Universal Robots PolyScope program: ur_comm_test.urp

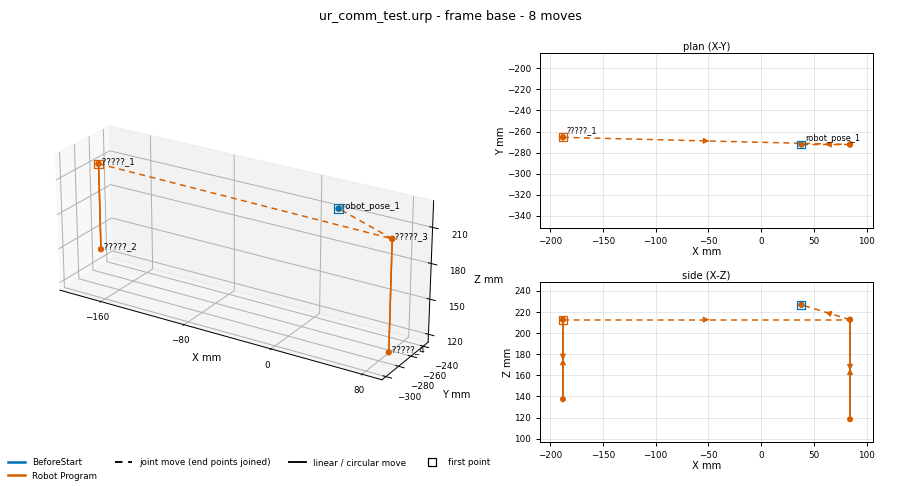
[picture p0: tool path of ur_comm_test.urp in frame base, 8 of 8 moves have a stored position in this frame; points joined in program order, loops and branches not executed]
Program ur_comm_test (installation=default directory=/programs/usbdisk/zivid-python-test/ur_comm_test_sample createdIn=5.5.1 lastSavedIn=5.21.0 robotSerialNumber=20195300395)
Calibrated DH parameters: a=[-0.000108, -0.14067, -0.21248, -0.000061, -0.000086, 0]; d=[0.151815, 81.30975, -77.69219, -3.486516, 0.085386, 0.091974]; alpha=[1.569683, -0.002449, 0.004563, 1.571204, -1.571811, 0]; deltaTheta=[0, -0.955759, 1.033289, -0.077525, 0.000001, 0]
InitVariablesNode
BeforeStart
  MoveJ speed 15 deg/s, acceleration 15 deg/s^2 (useActiveTCP=true optimoveEnabled=false optiMoveSpeed=0.3 optiMoveAcceleration=0.09) feature=Base
    Waypoint robot_pose_1: TCP in base x=38.181 y=-272.345 z=226.776 mm, rx=-2.0974 ry=2.253 rz=0.0086 rad; joints [-53.954, -85.282, -75.994, -109.42, 93.764, -49.87] deg; TCP offset x=-7.625 y=23.932 z=143.735 mm, rx=0 ry=0 rz=0 rad
  Script: write_output_integer_register(24,0)
  Script: write_output_boolean_register(64,False)
Robot Program (runOnlyOnce=false)
  Wait Condition expression=read_input_boolean_register(65)
  Script: write_output_integer_register(24,1)
  Script: write_output_boolean_register(64,True)
  Script: read_input_boolean_register(65)
  MoveJ speed 60 deg/s, acceleration 80 deg/s^2 (useActiveTCP=true optimoveEnabled=false optiMoveSpeed=0.3 optiMoveAcceleration=0.09) feature=Base
    Waypoint 웨이포인트_1: TCP in base x=-187.838 y=-265.519 z=212.755 mm, rx=2.1895 ry=-2.2511 rz=-0.0019 rad; joints [-96.693, -89.798, -75.994, -104.138, 90.098, -95.082] deg
  MoveL speed 250 mm/s, acceleration 1200 mm/s^2 (useActiveTCP=true optimoveEnabled=false optiMoveSpeed=0.3 optiMoveAcceleration=0.09) feature=Base
    Waypoint 웨이포인트_2: TCP in base x=-187.838 y=-265.519 z=137.312 mm, rx=2.1895 ry=-2.2511 rz=-0.0019 rad; joints [-96.737, -88.533, -97.686, -83.71, 90.113, -95.032] deg
    Waypoint 웨이포인트_1: TCP in base x=-187.838 y=-265.519 z=212.755 mm, rx=2.1895 ry=-2.2511 rz=-0.0019 rad; joints [-96.693, -89.798, -75.994, -104.138, 90.098, -95.082] deg
  MoveJ speed 60 deg/s, acceleration 80 deg/s^2 (useActiveTCP=true optimoveEnabled=false optiMoveSpeed=0.3 optiMoveAcceleration=0.09) feature=Base
    Waypoint 웨이포인트_3: TCP in base x=84.262 y=-272.319 z=212.755 mm, rx=2.1895 ry=-2.2511 rz=-0.0019 rad; joints [-43.139, -85.133, -80.384, -104.498, 90.134, -41.521] deg
  MoveL speed 250 mm/s, acceleration 1200 mm/s^2 (useActiveTCP=true optimoveEnabled=false optiMoveSpeed=0.3 optiMoveAcceleration=0.09) feature=Base
    Waypoint 웨이포인트_4: TCP in base x=84.262 y=-272.319 z=118.312 mm, rx=2.1895 ry=-2.2511 rz=-0.0019 rad; joints [-43.192, -84.436, -106.629, -78.949, 90.148, -41.458] deg
    Waypoint 웨이포인트_3: TCP in base x=84.262 y=-272.319 z=212.755 mm, rx=2.1895 ry=-2.2511 rz=-0.0019 rad; joints [-43.139, -85.133, -80.384, -104.498, 90.134, -41.521] deg
  Wait Sleep waitTime=0.5
  Script: write_output_integer_register(24,-1)
  MoveJ speed 15 deg/s, acceleration 15 deg/s^2 (useActiveTCP=true optimoveEnabled=false optiMoveSpeed=0.3 optiMoveAcceleration=0.09) feature=Base
    Waypoint robot_pose_1: TCP in base x=38.181 y=-272.345 z=226.776 mm, rx=-2.0974 ry=2.253 rz=0.0086 rad; joints [-53.954, -85.282, -75.994, -109.42, 93.764, -49.87] deg
  Halt
